PROGRAM PRG_ExitConvetor
VAR
	intnFBMotor : FB_Motors;
	intnFBIntlk : FB_Intlk;
END_VAR

intnFBIntlk (
	BackwardsInterlock01 := TRUE,
	BackwardsInterlock02 := TRUE,
	BackwardsInterlock03 := TRUE,
	BackwardsInterlock04 := TRUE,
	BackwardsInterlock05 := TRUE,
	ForwardInterlock01 := TRUE,
	ForwardInterlock02 := TRUE,
	ForwardInterlock03 := TRUE,
	ForwardInterlock04 := TRUE,
	ForwardInterlock05 := TRUE,
	oStsInterlockOK => intnFBMotor.inIntlkOK,
);

intnFBMotor (
	inStart := GVL.StartMachine,
	outOTE => Exit_Conveyor,
);

END_PROGRAM

(* stored: Version 1.1.0.1
   POU PRG_ExitConvetor: Id {2d4074f6-194d-4b9e-9de3-2585b363746c}, SpecialFunc None *)
